(* PLC project prj, KAIST_DSLAB noNameNow 1, author bwkim *)
(* stored: creationDateTime 2015-8-26T05:06:48, modificationDateTime 2015-8-26T05:06:48 *)

PROGRAM program3____HB
  VAR
    HB_CTUD : null;
  END_VAR
  VAR
    HB_CTUD_copy : null;
  END_VAR
  VAR_INPUT
    HB : INT;
  END_VAR
  VAR_OUTPUT
    HB_t0 : INT;
  END_VAR
  VAR  (* added by the conversion: wires and edge detectors of the diagram *)
    _LE_DINT11_OUT : INT;
    _OR3_BOOL25_OUT : BOOL;
  END_VAR

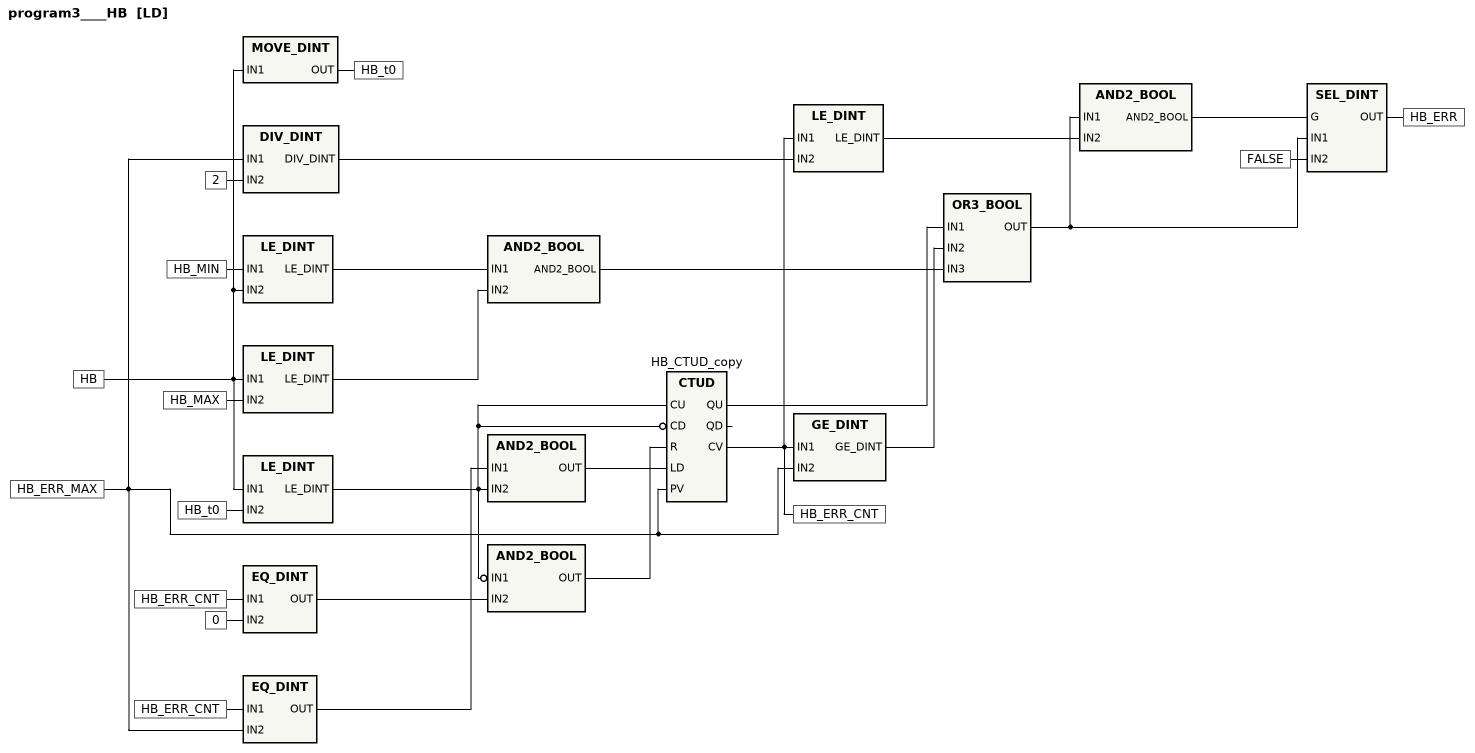
(* LD diagram, written out as Structured Text *)
HB_t0 := MOVE_DINT(HB);
_LE_DINT11_OUT := LE_DINT(HB, HB_t0);
HB_CTUD_copy(CU := _LE_DINT11_OUT, CD := NOT _LE_DINT11_OUT, R := AND2_BOOL(NOT _LE_DINT11_OUT, EQ_DINT(HB_ERR_CNT, 0)), LD := AND2_BOOL(EQ_DINT(HB_ERR_CNT, HB_ERR_MAX), _LE_DINT11_OUT), PV := HB_ERR_MAX);
HB_ERR_CNT := HB_CTUD_copy.CV;
_OR3_BOOL25_OUT := OR3_BOOL(HB_CTUD_copy.QU, GE_DINT(HB_CTUD_copy.CV, HB_ERR_MAX), AND2_BOOL(LE_DINT(HB_MIN, HB), LE_DINT(HB, HB_MAX)));
HB_ERR := SEL_DINT(AND2_BOOL(_OR3_BOOL25_OUT, LE_DINT(HB_CTUD_copy.CV, DIV_DINT(HB_ERR_MAX, 2))), _OR3_BOOL25_OUT, FALSE);
END_PROGRAM
